FUNCTION_BLOCK FB_BHKW
VAR
	Zustandscheck: FB_BHKW_Zustandscheck;
	Logik: FB_BHKW_Logik;
	Ablaufsteuerung: FB_BHKW_Ablaufsteuerung;
	Sollwertscheck: FB_BHKW_Sollwertscheck;
	Regelung: FB_BHKW_Regelung;
	Stellwertscheck: FB_BHKW_Stellwertscheck;
	QuitTrig: FB_SetResetFallTrigger;
	SchreibeDaten: FB_BHKW_Output;
	IN_Sammelstoerung AT %I* : BOOL;
	OUT_Betrieb AT %Q* : BOOL;
	OUT_Leistung AT %Q* : INT;
	LeseDaten: FB_BHKW_Modbus;
	Timer_freigabe: TOF;
END_VAR
VAR_INPUT
	Freigabe_auto: BOOL;
	Freigabe_Deakt_auto: BOOL;
	Betrieb_Anford_auto: BOOL;
	Regelung_Modus_auto: SINT;
	Regelung_Sollw_auto: REAL;
	Quittierung: BOOL;
	Adresse: STRING(15); (* IPv4 address of the target device *)
	BHKW_1_2: BOOL; (* False = BHKW1, True = BHKW2 *)
	Parameter_init: ST_BHKW_Parameter;
	Zustand_Pumpe: ST_PU_Zustand; (* Zustände der Pumpe auslesen, da Kommunikationsmodul nicht funktional *)
END_VAR
VAR_OUTPUT
	{attribute 'OPC.UA.DA' := '1'}Steuerung: ST_BHKW_Steuerung;
	{attribute 'OPC.UA.DA' := '1'}Stellwert: ST_BHKW_Stellwert;
	{attribute 'OPC.UA.DA' := '1'}Zustand: ST_BHKW_Zustand; 
	{attribute 'OPC.UA.DA' := '1'}Parameter: ST_BHKW_Parameter;
END_VAR
VAR // added by the converter: edge detectors and wires of the graphical bodies
    _w1, _w3, _w4 : BOOL;
    _w2 : ANY;
END_VAR

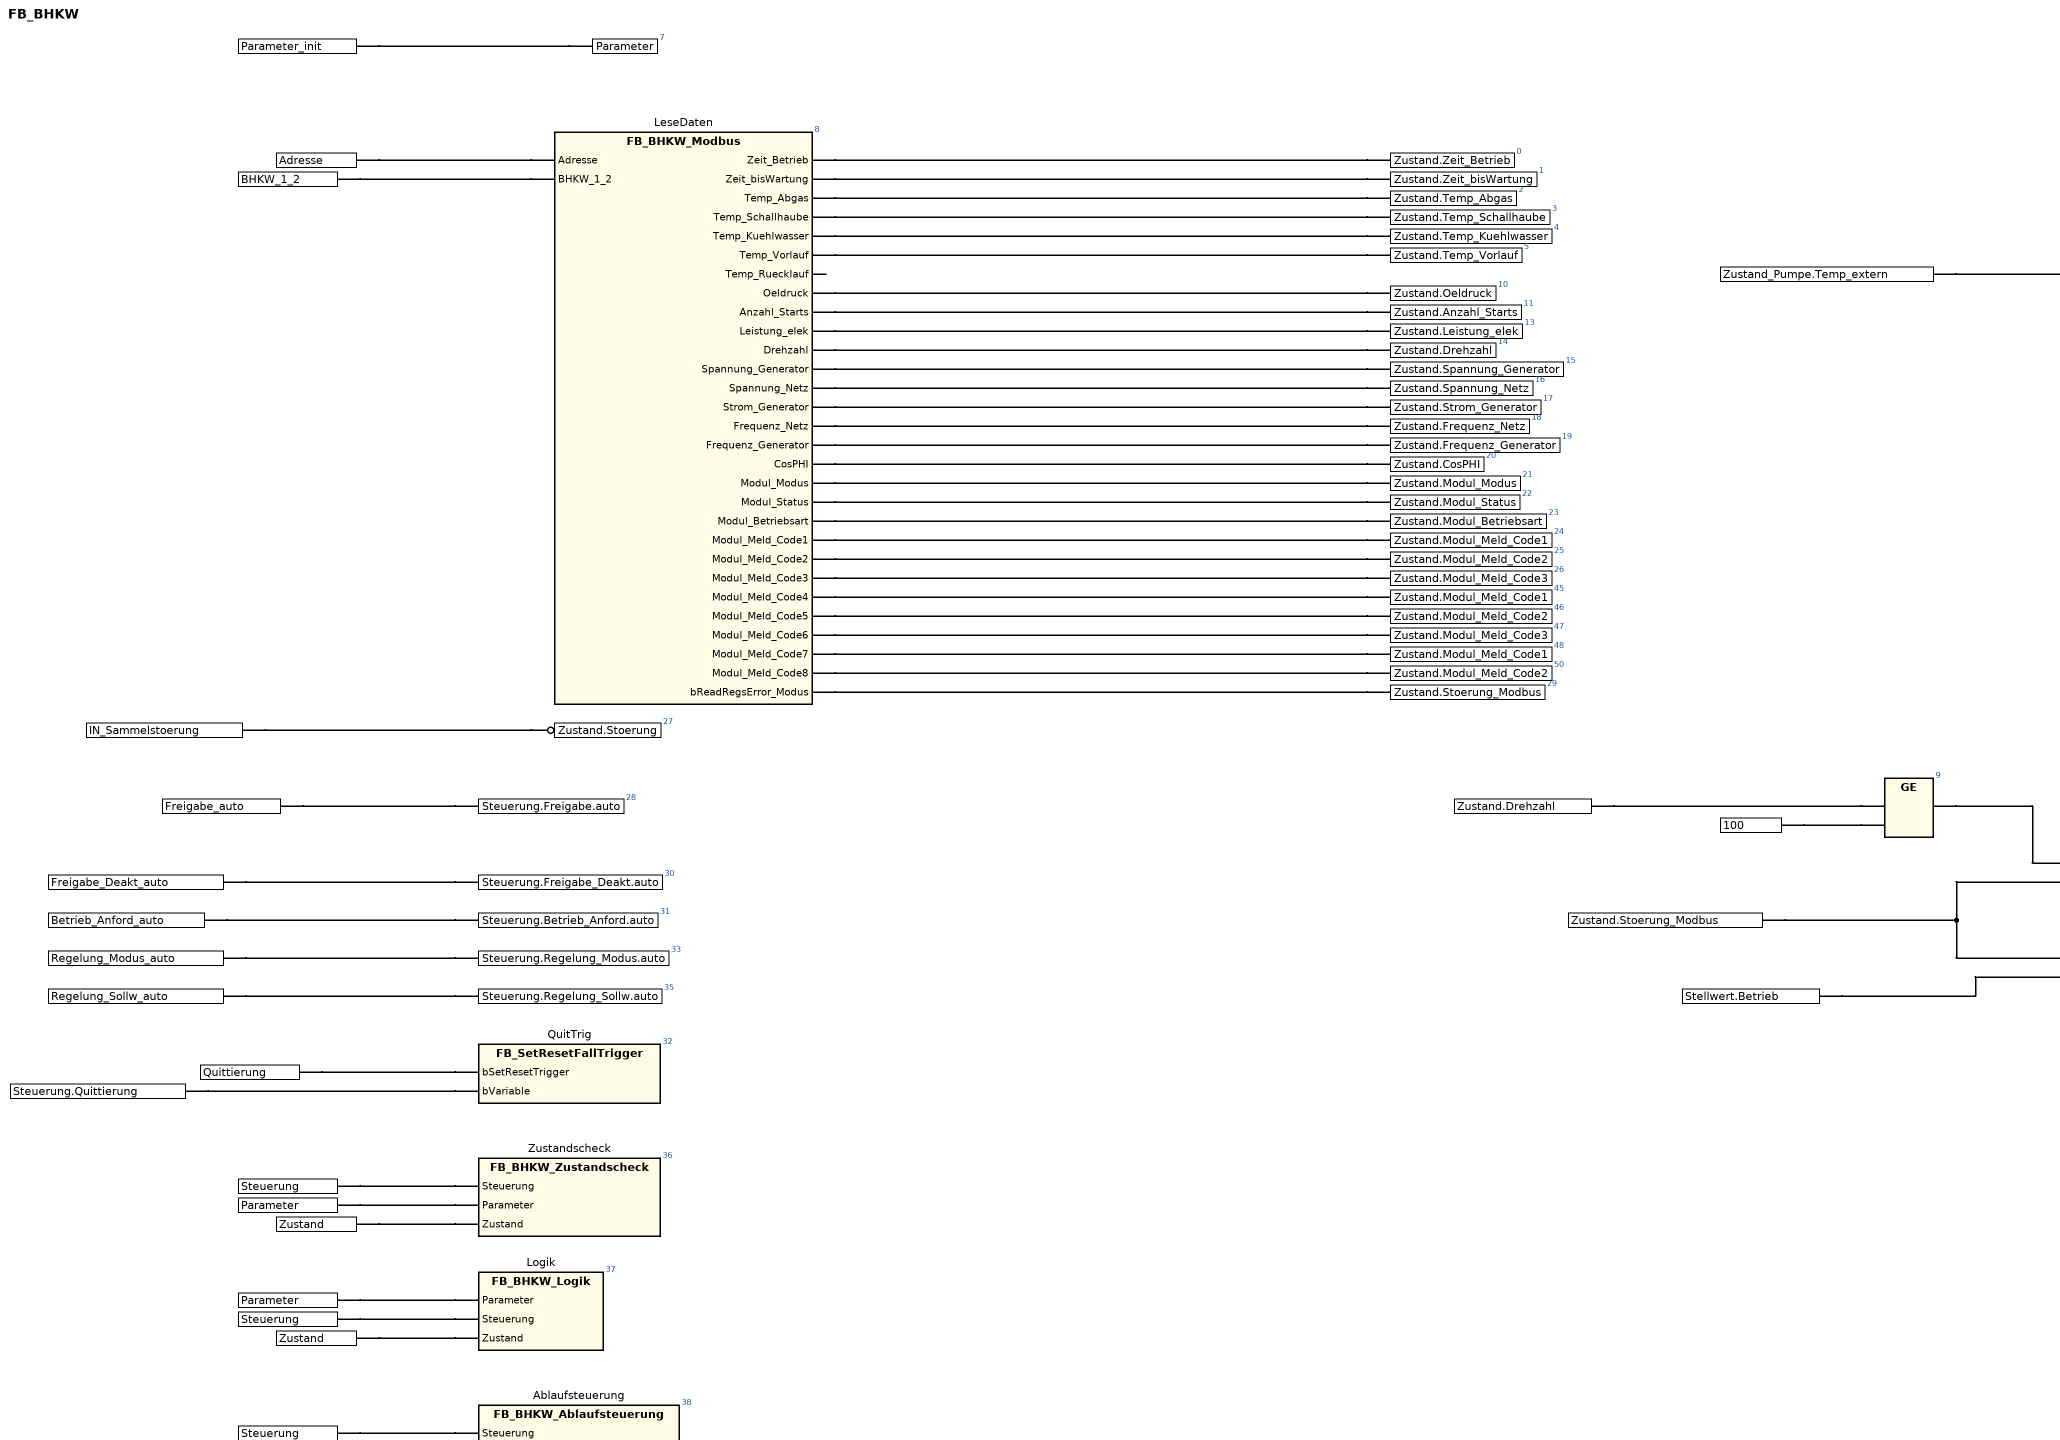
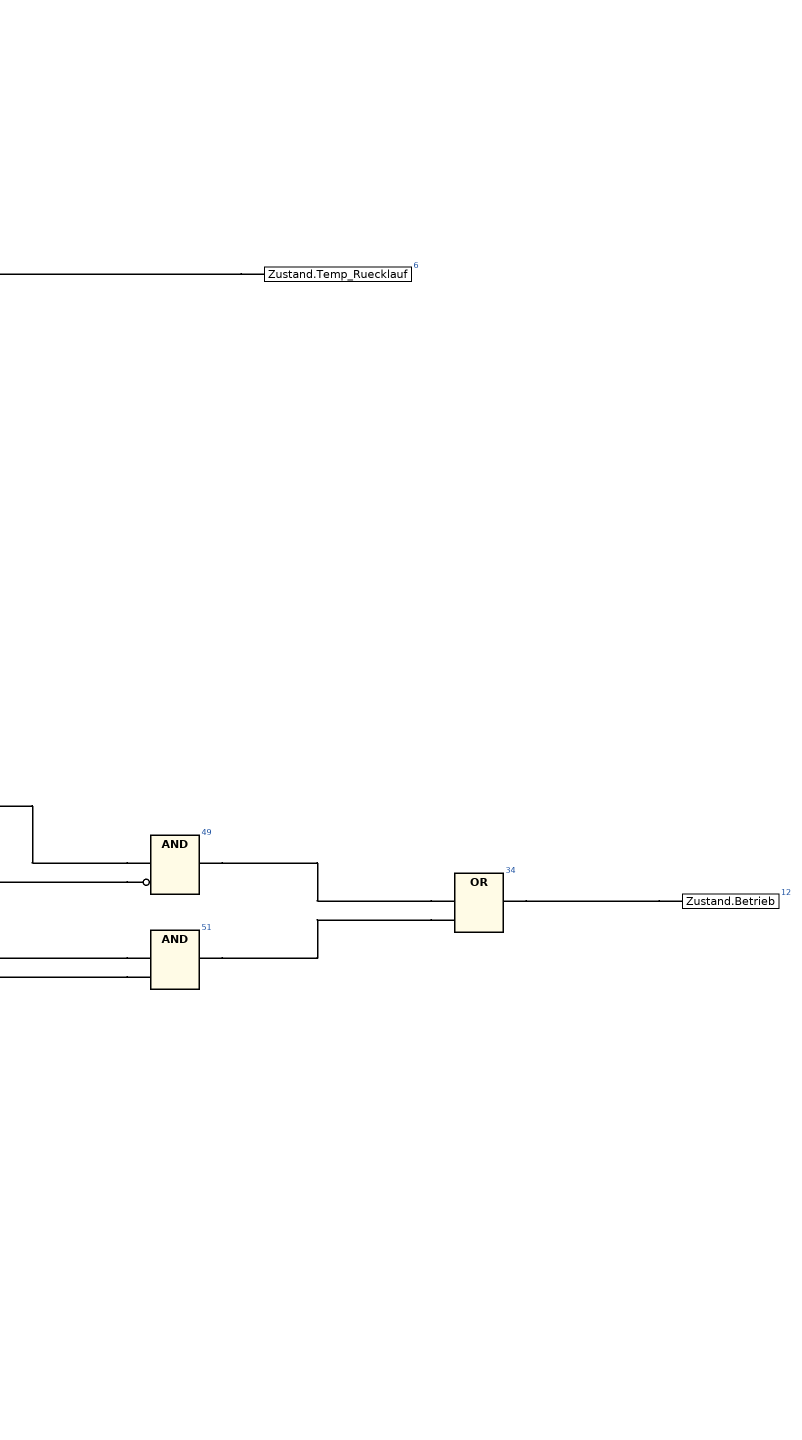
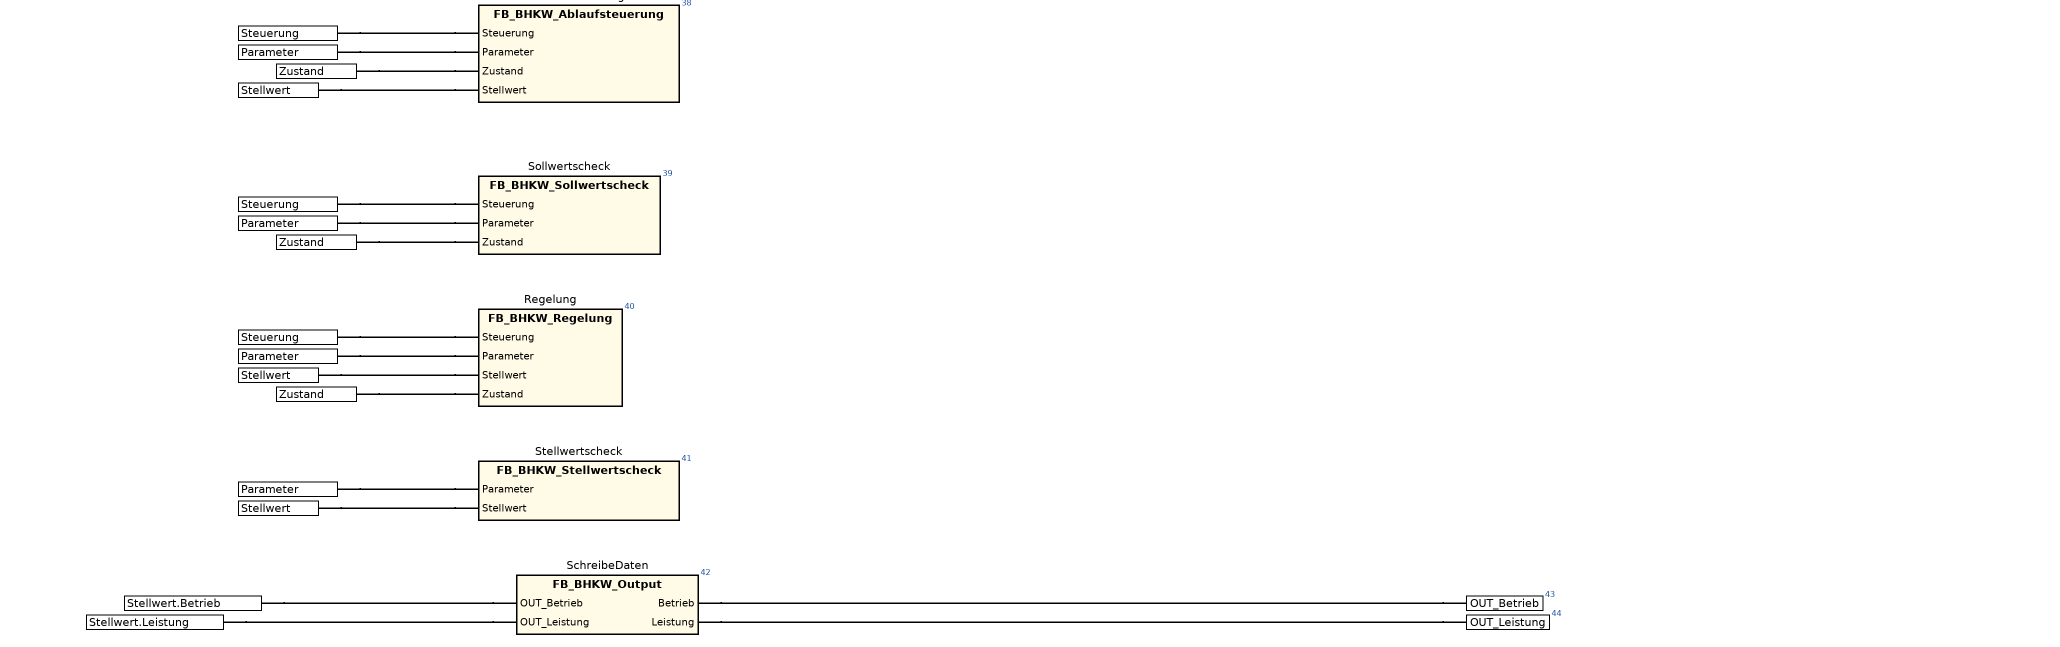
Zustand.Zeit_Betrieb := LeseDaten.Zeit_Betrieb;
Zustand.Zeit_bisWartung := LeseDaten.Zeit_bisWartung;
Zustand.Temp_Abgas := LeseDaten.Temp_Abgas;
Zustand.Temp_Schallhaube := LeseDaten.Temp_Schallhaube;
Zustand.Temp_Kuehlwasser := LeseDaten.Temp_Kuehlwasser;
Zustand.Temp_Vorlauf := LeseDaten.Temp_Vorlauf;
Zustand.Temp_Ruecklauf := Zustand_Pumpe.Temp_extern;
Parameter := Parameter_init;
LeseDaten(Adresse := Adresse, BHKW_1_2 := BHKW_1_2); // FB_BHKW_Modbus
_w1 := Zustand.Drehzahl >= 100;
Zustand.Oeldruck := LeseDaten.Oeldruck;
Zustand.Anzahl_Starts := LeseDaten.Anzahl_Starts;
Zustand.Betrieb := _w2;
Zustand.Leistung_elek := LeseDaten.Leistung_elek;
Zustand.Drehzahl := LeseDaten.Drehzahl;
Zustand.Spannung_Generator := LeseDaten.Spannung_Generator;
Zustand.Spannung_Netz := LeseDaten.Spannung_Netz;
Zustand.Strom_Generator := LeseDaten.Strom_Generator;
Zustand.Frequenz_Netz := LeseDaten.Frequenz_Netz;
Zustand.Frequenz_Generator := LeseDaten.Frequenz_Generator;
Zustand.CosPHI := LeseDaten.CosPHI;
Zustand.Modul_Modus := LeseDaten.Modul_Modus;
Zustand.Modul_Status := LeseDaten.Modul_Status;
Zustand.Modul_Betriebsart := LeseDaten.Modul_Betriebsart;
Zustand.Modul_Meld_Code1 := LeseDaten.Modul_Meld_Code1;
Zustand.Modul_Meld_Code2 := LeseDaten.Modul_Meld_Code2;
Zustand.Modul_Meld_Code3 := LeseDaten.Modul_Meld_Code3;
Zustand.Stoerung := NOT IN_Sammelstoerung;
Steuerung.Freigabe.auto := Freigabe_auto;
Zustand.Stoerung_Modbus := LeseDaten.bReadRegsError_Modus;
Steuerung.Freigabe_Deakt.auto := Freigabe_Deakt_auto;
Steuerung.Betrieb_Anford.auto := Betrieb_Anford_auto;
QuitTrig(bSetResetTrigger := Quittierung, bVariable := Steuerung.Quittierung); // FB_SetResetFallTrigger
Steuerung.Regelung_Modus.auto := Regelung_Modus_auto;
_w2 := _w3 OR _w4;
Steuerung.Regelung_Sollw.auto := Regelung_Sollw_auto;
Zustandscheck(Steuerung := Steuerung, Parameter := Parameter, Zustand := Zustand); // FB_BHKW_Zustandscheck
Logik(Parameter := Parameter, Steuerung := Steuerung, Zustand := Zustand); // FB_BHKW_Logik
Ablaufsteuerung(Steuerung := Steuerung, Parameter := Parameter, Zustand := Zustand, Stellwert := Stellwert); // FB_BHKW_Ablaufsteuerung
Sollwertscheck(Steuerung := Steuerung, Parameter := Parameter, Zustand := Zustand); // FB_BHKW_Sollwertscheck
Regelung(Steuerung := Steuerung, Parameter := Parameter, Stellwert := Stellwert, Zustand := Zustand); // FB_BHKW_Regelung
Stellwertscheck(Parameter := Parameter, Stellwert := Stellwert); // FB_BHKW_Stellwertscheck
SchreibeDaten(OUT_Betrieb := Stellwert.Betrieb, OUT_Leistung := Stellwert.Leistung); // FB_BHKW_Output
OUT_Betrieb := SchreibeDaten.Betrieb;
OUT_Leistung := SchreibeDaten.Leistung;
Zustand.Modul_Meld_Code1 := LeseDaten.Modul_Meld_Code4;
Zustand.Modul_Meld_Code2 := LeseDaten.Modul_Meld_Code5;
Zustand.Modul_Meld_Code3 := LeseDaten.Modul_Meld_Code6;
Zustand.Modul_Meld_Code1 := LeseDaten.Modul_Meld_Code7;
_w3 := _w1 AND NOT Zustand.Stoerung_Modbus;
Zustand.Modul_Meld_Code2 := LeseDaten.Modul_Meld_Code8;
_w4 := Zustand.Stoerung_Modbus AND Stellwert.Betrieb;

END_FUNCTION_BLOCK

(* stored: Version 1.1.0.1, ProductVersion 3.1.4024.9
   POU FB_BHKW: Id {6299133a-97c8-4146-a814-0e07582dc10a}, SpecialFunc None *)
